TYPE E_MachineMode :
(
	UNDEFINE := 0,
	MANUAL	:=1		  ,
	AUTO	:=2		  ,
	SERVICE :=3,
	ModeSelect:=99
)INT;
END_TYPE

(* stored: Version 1.1.0.1, ProductVersion 3.1.4024.13
   DUT E_MachineMode: Id {5f4649af-d81d-4702-a7c7-15f8c775ae27} *)
